TYPE MNG_DatagramHeader :
STRUCT
	/// Time when datagram has been created 
	Counter: DWORD;
	/// Time when datagram has been sent 
	SentTime: DWORD;
	/// Type of the datagram 
	DatagramType: DWORD := MNG_UnknownDatagram;
	/// Byte count in the payload 
	ByteCount: DWORD := 0;
END_STRUCT
END_TYPE

(* stored: Version 1.1.0.1, ProductVersion 3.1.0.25
   DUT MNG_DatagramHeader: Id {ea2ec010-a730-499f-977c-c8d4af337a98} *)
